INTERFACE I_HaveExtensions EXTENDS __SYSTEM.IQueryInterface

METHOD AddExtension
VAR_INPUT
	ExtensionToAdd : I_Extension;
END_VAR
END_METHOD

METHOD PUBLIC GetExtensions : I_ExtensionCollection
VAR_INPUT
END_VAR
END_METHOD

METHOD PUBLIC TryGetExtensionByName : BOOL
VAR_INPUT
	Name : T_MAXSTRING;
	Destination : REFERENCE TO I_Extension;
END_VAR
END_METHOD

END_INTERFACE

(* stored: Version 1.1.0.1, ProductVersion 3.1.4024.12
   Itf I_HaveExtensions: Id {2c4d3330-a4d5-0bf1-1982-102b528ecb24}
   Method AddExtension: Id {21dfd60d-3eac-0633-1fbc-e2a67a4a7248}
   Method GetExtensions: Id {ded8e208-00db-0046-2018-6597a6e965e4}
   Method TryGetExtensionByName: Id {6387349c-8660-06ad-3b9d-60ffa3ef67c8} *)
